INTERFACE I_StateMachine EXTENDS Debug.I_Debug, Tags.I_Tagged

METHOD ChangeState : Results.Result
VAR_INPUT
	iNewState	: I_State;
END_VAR
VAR_OUTPUT
	iOldState	: I_State;
END_VAR
END_METHOD

METHOD GetState : I_State
VAR_INPUT
END_VAR
END_METHOD

END_INTERFACE

(* stored: Version 1.1.0.1
   Itf I_StateMachine: Id {848c5871-668a-436e-b188-ec716f6b51de}
   Method ChangeState: Id {aa325f6c-21a2-4331-a99e-3f4622014108}
   Method GetState: Id {19136f5c-d84a-49bd-8f73-9efae45b8ecd} *)
